// TIA Portal V18 export
FUNCTION "AHUModePanelSwitch" : Void   // FC60101, LAD
{ S7_Optimized_Access := 'TRUE' }
VERSION : 0.1
// stored: AutoNumber false, IsIECCheckEnabled false, SetENOAutomatically false, UDAEnableTagReadback false
   VAR_INPUT
      iUnitID : Int;
      xPanelSelectorOff : Bool;
      xPanelSelector1Sp : Bool;
      xPanelSelector2Sp : Bool;
      xPanelSelectorAuto : Bool;
   END_VAR
   VAR_OUTPUT
      cPanelSelectorState : Byte;
   END_VAR
BEGIN

REGION Network 1 (SCL)
   IF #xPanelSelectorOff THEN
       #cPanelSelectorState := 0;//Off
   ELSIF #xPanelSelector1Sp THEN
       #cPanelSelectorState := 2;//Speed1
   ELSIF #xPanelSelector2Sp THEN
       #cPanelSelectorState := 3;//Speed2
   ELSE
       #cPanelSelectorState := 4;//Auto
   END_IF;
END_REGION
END_FUNCTION
